// PLC global variables
{attribute 'qualified_only'}
VAR_GLOBAL
    AMSNetId AT %I* : AMSNETID;
END_VAR

(* stored: Version 1.1.0.1, ProductVersion 3.1.4024.6
   GVL GVL_PLC: Id {539a127c-f7fe-4875-9bf7-a09bc28f6f17} *)
